// TIA Portal V17 export
// export: Created 2025-03-12T15:33:07.5470294Z, ExportSetting WithDefaults, DisplayName Totally Integrated Automation Portal, DisplayVersion V17 Update 8, DisplayName TIA Portal Openness, DisplayVersion V17 Update 8, DisplayName TIA Portal Version Control Interface, DisplayVersion V17, DisplayName SINAMICS Startdrive Advanced, DisplayVersion V17 SP2, DisplayName SINAMICS Startdrive G110M, G120, G120C, G120D, G120P, G115D, DisplayVersion V17 SP2, DisplayName SINAMICS Startdrive G130, G150, S120, S150, SINAMICS MV, S210, DisplayVersion V17 SP2, DisplayName STEP 7 Professional, DisplayVersion V17 Update 8, DisplayName SINUMERIK ONE STEP 7 Toolbox, DisplayVersion V17 Update 12, DisplayName SINUMERIK 840D sl STEP 7 Toolbox, DisplayVersion V17 Update 12, DisplayName STEP 7 Safety, DisplayVersion V17 Update 6, DisplayName WinCC Advanced, DisplayVersion V17 Update 8
FUNCTION_BLOCK "FB1031_BRAKE_TEST"   // FB1031, LAD
{ S7_Optimized_Access := 'FALSE' }
AUTHOR : ETXETAR
VERSION : 1.0
// stored: AutoNumber false, IsIECCheckEnabled false, SetENOAutomatically false, UDAEnableTagReadback false
   VAR_INPUT
      START_REQ : Bool;   // REQUEST FOR START BRAKE TEST / START REQUEST
      BRAKE_SELECT : Bool;   // Selection of brake 1 or 2 - set to 0 for brake 1, set to 1for brake 2. / BRAKE SELECTION
      DIRECTION_OF_ROT : Bool;   // Direction of rotation - set to 0 for positive, set to 1 fornegative. / DIRECTION OF ROTATION
      TORQUE_SELECT : Bool;   // Torque 1 or 2 - set to 0 for Test torquefactor 1, set to 1for Test torquefactor 2. / TORQUE SELECTION
      "BRAKE_CLOSED(ONLY EXTERNAL)" : Bool;   // Brake closed - Set to 1 to confirm that the brake isclosed (External brakes only) / BRAKE CLOSED(ONLY EXTERNAL)
   END_VAR
   VAR_OUTPUT
      BRAKE_TEST_ACTIVE : Bool;   // Brake test is active - 1 = brake test active. / BRAKE TEST ACTIVE
      BRAKE_TEST_DONE : Bool;   // Brake test ok - 1 = brake test was successful. / BRAKE TEST DONE
      BRAKE_TEST_ERROR : Bool;   // Brake test nok - 1 = brake test was NOT successful. / BRAKE TEST ERROR
      SELECTED_BRAKE : Bool;   // Brake 1 or 2 active - 0 = brake 1, 1 = brake 2. / SELECTED BRAKE
      "BRAKE_REQ(ONLY_EXTERNAL)" : Bool;   // Close brake request for external brakes / BRAKE REQ(ONLY EXTERNAL)
      SIGN_OF_LOAD : Bool;   // Load torque sign - direction of the load torque,0 = positive, 1 = negative. Can be used to determinethe SBT direction. / SIGN OF LOAD
   END_VAR
   VAR_IN_OUT
      AXIS_DB : "LBP_typeAxisX";
   END_VAR
   VAR DB_SPECIFIC
      Timer_Brake_test_DONE { ExternalAccessible := 'False'; ExternalVisible := 'False'; ExternalWritable := 'False'; S7_SetPoint := 'True'} : TON_TIME;
      Timer_Brake_test_ERROR { ExternalAccessible := 'False'; ExternalVisible := 'False'; ExternalWritable := 'False'; S7_SetPoint := 'True'} : TON_TIME;
   END_VAR
BEGIN

REGION Network 1: BRAKE SELECTION / Test con freno 1 o 2
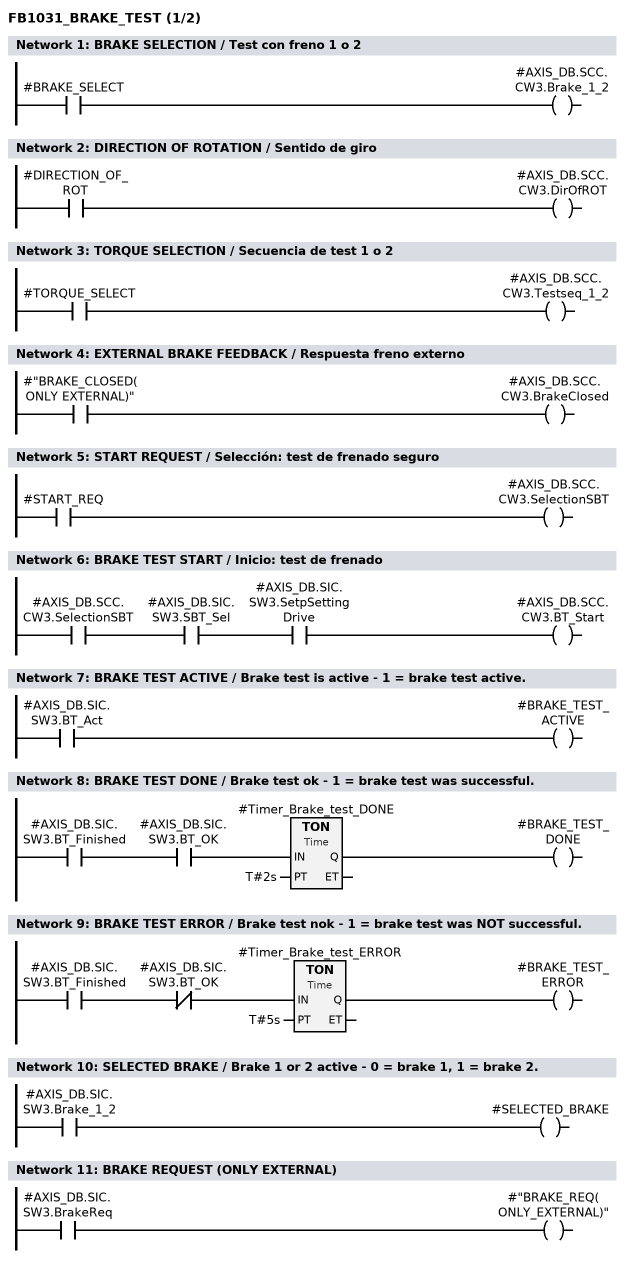
   RUNG wire#powerrail
      Contact( #BRAKE_SELECT )
      Coil( #AXIS_DB.SCC.CW3.Brake_1_2 )
   END_RUNG
   // the same network as SCL:
   #AXIS_DB.SCC.CW3.Brake_1_2 := #BRAKE_SELECT;
END_REGION

REGION Network 2: DIRECTION OF ROTATION / Sentido de giro
   RUNG wire#powerrail
      Contact( #DIRECTION_OF_ROT )
      Coil( #AXIS_DB.SCC.CW3.DirOfROT )
   END_RUNG
   // the same network as SCL:
   #AXIS_DB.SCC.CW3.DirOfROT := #DIRECTION_OF_ROT;
END_REGION

REGION Network 3: TORQUE SELECTION / Secuencia de test 1 o 2
   RUNG wire#powerrail
      Contact( #TORQUE_SELECT )
      Coil( #AXIS_DB.SCC.CW3.Testseq_1_2 )
   END_RUNG
   // the same network as SCL:
   #AXIS_DB.SCC.CW3.Testseq_1_2 := #TORQUE_SELECT;
END_REGION

REGION Network 4: EXTERNAL BRAKE FEEDBACK / Respuesta freno externo
   RUNG wire#powerrail
      Contact( #"BRAKE_CLOSED(ONLY EXTERNAL)" )
      Coil( #AXIS_DB.SCC.CW3.BrakeClosed )
   END_RUNG
   // the same network as SCL:
   #AXIS_DB.SCC.CW3.BrakeClosed := #"BRAKE_CLOSED(ONLY EXTERNAL)";
END_REGION

REGION Network 5: START REQUEST / Selección: test de frenado seguro
   RUNG wire#powerrail
      Contact( #START_REQ )
      Coil( #AXIS_DB.SCC.CW3.SelectionSBT )
   END_RUNG
   // the same network as SCL:
   #AXIS_DB.SCC.CW3.SelectionSBT := #START_REQ;
END_REGION

REGION Network 6: BRAKE TEST START / Inicio: test de frenado
   RUNG wire#powerrail
      Contact( #AXIS_DB.SCC.CW3.SelectionSBT )
      Contact( #AXIS_DB.SIC.SW3.SBT_Sel )
      Contact( #AXIS_DB.SIC.SW3.SetpSettingDrive )
      Coil( #AXIS_DB.SCC.CW3.BT_Start )
   END_RUNG
   // the same network as SCL:
   #AXIS_DB.SCC.CW3.BT_Start := #AXIS_DB.SCC.CW3.SelectionSBT AND #AXIS_DB.SIC.SW3.SBT_Sel AND #AXIS_DB.SIC.SW3.SetpSettingDrive;
END_REGION

REGION Network 7: BRAKE TEST ACTIVE / Brake test is active - 1 = brake test active.
   RUNG wire#powerrail
      Contact( #AXIS_DB.SIC.SW3.BT_Act )
      Coil( #BRAKE_TEST_ACTIVE )
   END_RUNG
   // the same network as SCL:
   #BRAKE_TEST_ACTIVE := #AXIS_DB.SIC.SW3.BT_Act;
END_REGION

REGION Network 8: BRAKE TEST DONE / Brake test ok - 1 = brake test was successful.
   RUNG wire#powerrail
      Contact( #AXIS_DB.SIC.SW3.BT_Finished )
      Contact( #AXIS_DB.SIC.SW3.BT_OK )
      { S7_Templates := "time_type := Time" } #Timer_Brake_test_DONE.TON(pt := T#2s, et =>)
      Coil( #BRAKE_TEST_DONE )
   END_RUNG
   // the same network as SCL:
   #Timer_Brake_test_DONE(IN := #AXIS_DB.SIC.SW3.BT_Finished AND #AXIS_DB.SIC.SW3.BT_OK, PT := T#2s);   // TON
   #BRAKE_TEST_DONE := #Timer_Brake_test_DONE.Q;
END_REGION

REGION Network 9: BRAKE TEST ERROR / Brake test nok - 1 = brake test was NOT successful.
   RUNG wire#powerrail
      Contact( #AXIS_DB.SIC.SW3.BT_Finished )
      I_Contact( #AXIS_DB.SIC.SW3.BT_OK )
      { S7_Templates := "time_type := Time" } #Timer_Brake_test_ERROR.TON(pt := T#5s, et =>)
      Coil( #BRAKE_TEST_ERROR )
   END_RUNG
   // the same network as SCL:
   #Timer_Brake_test_ERROR(IN := #AXIS_DB.SIC.SW3.BT_Finished AND NOT #AXIS_DB.SIC.SW3.BT_OK, PT := T#5s);   // TON
   #BRAKE_TEST_ERROR := #Timer_Brake_test_ERROR.Q;
END_REGION

REGION Network 10: SELECTED BRAKE / Brake 1 or 2 active - 0 = brake 1, 1 = brake 2.
   RUNG wire#powerrail
      Contact( #AXIS_DB.SIC.SW3.Brake_1_2 )
      Coil( #SELECTED_BRAKE )
   END_RUNG
   // the same network as SCL:
   #SELECTED_BRAKE := #AXIS_DB.SIC.SW3.Brake_1_2;
END_REGION

REGION Network 11: BRAKE REQUEST (ONLY EXTERNAL)
   RUNG wire#powerrail
      Contact( #AXIS_DB.SIC.SW3.BrakeReq )
      Coil( #"BRAKE_REQ(ONLY_EXTERNAL)" )
   END_RUNG
   // the same network as SCL:
   #"BRAKE_REQ(ONLY_EXTERNAL)" := #AXIS_DB.SIC.SW3.BrakeReq;
END_REGION

REGION Network 12: SIGN OF LOAD / Load torque sign - direction of the load torque,0 = positive, 1 = negative. Can be used to determinethe SBT direction.
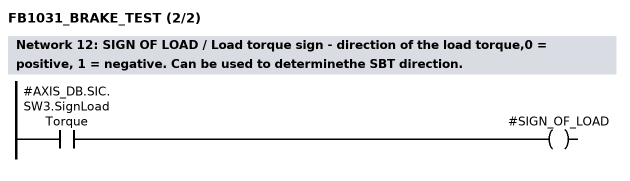
   RUNG wire#powerrail
      Contact( #AXIS_DB.SIC.SW3.SignLoadTorque )
      Coil( #SIGN_OF_LOAD )
   END_RUNG
   // the same network as SCL:
   #SIGN_OF_LOAD := #AXIS_DB.SIC.SW3.SignLoadTorque;
END_REGION
END_FUNCTION_BLOCK
